// TwinCAT 3 PLC project PLC
// ProgramVersion: 3.1.4023.0
// libraries:
//   Tc2_Standard, * (Beckhoff Automation GmbH)
//   Tc2_System, * (Beckhoff Automation GmbH)
//   Tc3_Module, * (Beckhoff Automation GmbH)
// project tree:
//   / CheckPointer.TcPOU, Examples.TcPOU, InterfaceExample.TcPOU, I_Interface.TcIO, PlcTask.TcTTO, PointerExample.TcPOU, ReferenceExample.TcPOU
// real-time tasks:
//   TASK PlcTask: cycle T#10ms, priority 20, ADS port 350

CONFIGURATION PLC
    RESOURCE PLC ON TwinCAT3
        TASK PlcTask(INTERVAL := T#10ms, PRIORITY := 20);
        PROGRAM Examples WITH PlcTask : Examples;
    END_RESOURCE
END_CONFIGURATION

// ---- I_Interface.TcIO
INTERFACE I_Interface

PROPERTY SomeProperty : INT
GET
END_GET
SET
END_SET
END_PROPERTY

END_INTERFACE

// ---- Examples.TcPOU
PROGRAM Examples

//PointerExample();
//ReferenceExample();
InterfaceExample();

END_PROGRAM

// ---- InterfaceExample.TcPOU
PROGRAM InterfaceExample
VAR
    number : INT;
    someInterface : I_Interface;
END_VAR

//// This code causes a page fault
//number := someInterface.SomeProperty;

// This code doesn't cause a page fault
IF someInterface <> 0 THEN
    number := someInterface.SomeProperty;
END_IF

END_PROGRAM

// ---- CheckPointer.TcPOU
// Implicitly generated code : DO NOT EDIT
FUNCTION CheckPointer : POINTER TO BYTE
VAR_INPUT
    ptToTest : POINTER TO BYTE; // Destination address of the pointer
    iSize : DINT;		        // Size of the type the pointer points to. (e.g: 20 for POINTER TO ARRAY [0..9] OF INT)
    iGran : DINT;		        // Granularity of the pointer access. This is the size of the biggest non-structured data type in the type the pointer points to. (e.g: 2 for POINTER TO ARRAY [0..9] OF INT)
    bWrite: BOOL;		        // Indicates read or write Access. TRUE = write access.
END_VAR

// Implicitly generated code : Only an Implementation suggestion
{noflow}
IF ptToTest=0 THEN
    ADSLOGSTR(ADSLOG_MSGTYPE_ERROR OR ADSLOG_MSGTYPE_STRING,'CheckPointer failed due to invalid address.','');
ELSIF iSize<=0 THEN
    ADSLOGSTR(ADSLOG_MSGTYPE_ERROR OR ADSLOG_MSGTYPE_STRING,'CheckPointer failed due to invalid size.','');
ELSIF iGran<=0 THEN
    ADSLOGSTR(ADSLOG_MSGTYPE_ERROR OR ADSLOG_MSGTYPE_STRING,'CheckPointer failed due to invalid granularity.','');
// -> Please note that the following memory area check is time consuming:
//ELSIF F_CheckMemoryArea(pData:=ptToTest,nSize:=DINT_TO_UDINT(iSize)) = E_TcMemoryArea.Unknown THEN
//    ADSLOGSTR(ADSLOG_MSGTYPE_ERROR OR ADSLOG_MSGTYPE_STRING,'CheckPointer failed due to unknown memory area.','');
END_IF
CheckPointer := ptToTest;
{flow}

END_FUNCTION

// ---- PointerExample.TcPOU
PROGRAM PointerExample
VAR
    pointerToNumber : POINTER TO INT;
    number : INT;
END_VAR

// This code causes a page fault
number := pointerToNumber^;

// This code doesn't cause a page fault
IF pointerToNumber <> 0 THEN
    number := pointerToNumber^;
END_IF

END_PROGRAM

// ---- ReferenceExample.TcPOU
PROGRAM ReferenceExample
VAR
    refNumber : REFERENCE TO INT;
END_VAR

//// This causes a page fault
//refNumber := 1;

// This doesn't cause a page fault
IF __ISVALIDREF(refNumber) THEN
    refNumber := 1;
END_IF

END_PROGRAM
